SUBAPPLICATION Counter (* Subapplication Type *)
  (* Standard: 61499-2 *)
  (* Version 1.0, 2023-02-17, Franz *)
  IMPORT FBs::Counter::const::DefaultPool::AuxFunction2_MinusMinus;
  IMPORT FBs::Counter::const::DefaultPool::AuxFunction2_PlusPlus;
  IMPORT FBs::Counter::const::DefaultPool::Button_MinusMinus;
  IMPORT FBs::Counter::const::DefaultPool::Button_NextVT;
  IMPORT FBs::Counter::const::DefaultPool::Button_PlusPlus;
  IMPORT FBs::Counter::const::DefaultPool::Button_Reset_Gesamtzaehler;
  IMPORT FBs::Counter::const::DefaultPool::Button_Reset_Tageszaehler;
  IMPORT FBs::Counter::const::DefaultPool::NumberVariable_Gesamtzaehler;
  IMPORT FBs::Counter::const::DefaultPool::NumberVariable_Gesamtziel;
  IMPORT FBs::Counter::const::DefaultPool::NumberVariable_Tageszaehler;
  IMPORT FBs::Counter::const::DefaultPool::NumberVariable_Tagesziel;
  IMPORT FBs::Counter::const::DefaultPool::ObjectPointer_Gesamtziel;
  IMPORT FBs::Counter::const::DefaultPool::ObjectPointer_Tagesziel;
  IMPORT FBs::Counter::const::DefaultPool::SoftKey_MinusMinus;
  IMPORT FBs::Counter::const::DefaultPool::SoftKey_PlusPlus;
  IMPORT FBs::Counter::const::DefaultPool::SoftKey_Reset_Gesamtzaehler;
  IMPORT FBs::Counter::const::DefaultPool::SoftKey_Reset_Tageszaehler;
  IMPORT NVS_Keys::KEY_GESAMTZAEHLER;
  IMPORT NVS_Keys::KEY_GESAMTZIEL;
  IMPORT NVS_Keys::KEY_TAGESZAEHLER;
  IMPORT NVS_Keys::KEY_TAGESZIEL;
  IMPORT isobus::UT::io::Button::ButtonActivationCode::BT_RELEASED_UNLATCHED;
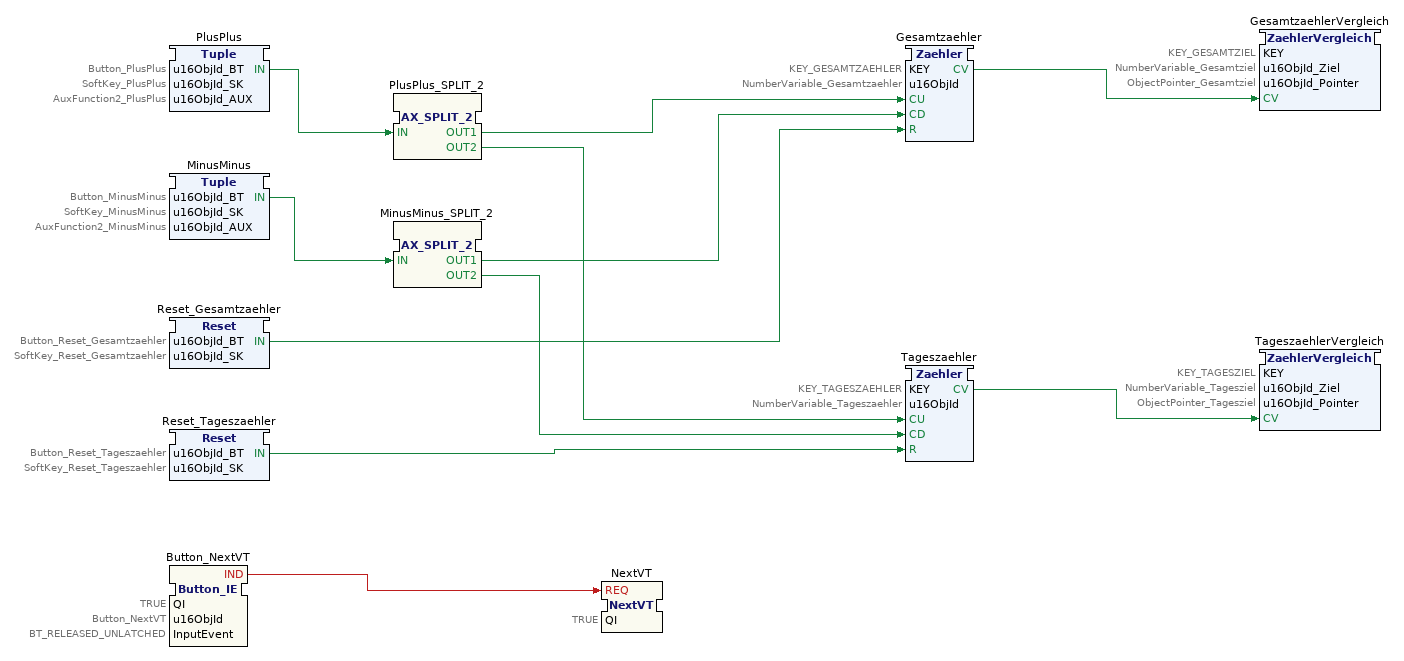
  FBS
    NextVT : isobus::UT::util::NextVT(QI := TRUE);
    Button_NextVT : isobus::UT::io::Button::Button_IE(QI := TRUE, u16ObjId := Button_NextVT, InputEvent := BT_RELEASED_UNLATCHED);
    PlusPlus_SPLIT_2 : adapter::events::unidirectional::AX_SPLIT_2;
    MinusMinus_SPLIT_2 : adapter::events::unidirectional::AX_SPLIT_2;
  END_FBS
  SUBAPPS
    MinusMinus : FBs::Counter::subs::Buttons::Tuple(u16ObjId_BT := Button_MinusMinus, u16ObjId_SK := SoftKey_MinusMinus, u16ObjId_AUX := AuxFunction2_MinusMinus);
    PlusPlus : FBs::Counter::subs::Buttons::Tuple(u16ObjId_BT := Button_PlusPlus, u16ObjId_SK := SoftKey_PlusPlus, u16ObjId_AUX := AuxFunction2_PlusPlus);
    Reset_Gesamtzaehler : FBs::Counter::subs::Buttons::Reset(u16ObjId_BT := Button_Reset_Gesamtzaehler, u16ObjId_SK := SoftKey_Reset_Gesamtzaehler);
    Reset_Tageszaehler : FBs::Counter::subs::Buttons::Reset(u16ObjId_BT := Button_Reset_Tageszaehler, u16ObjId_SK := SoftKey_Reset_Tageszaehler);
    Gesamtzaehler : FBs::Counter::subs::Zaehler::Zaehler(KEY := KEY_GESAMTZAEHLER, u16ObjId := NumberVariable_Gesamtzaehler);
    Tageszaehler : FBs::Counter::subs::Zaehler::Zaehler(KEY := KEY_TAGESZAEHLER, u16ObjId := NumberVariable_Tageszaehler);
    TageszaehlerVergleich : FBs::Counter::subs::Zaehler::ZaehlerVergleich(KEY := KEY_TAGESZIEL, u16ObjId_Ziel := NumberVariable_Tagesziel, u16ObjId_Pointer := ObjectPointer_Tagesziel);
    GesamtzaehlerVergleich : FBs::Counter::subs::Zaehler::ZaehlerVergleich(KEY := KEY_GESAMTZIEL, u16ObjId_Ziel := NumberVariable_Gesamtziel, u16ObjId_Pointer := ObjectPointer_Gesamtziel);
  END_SUBAPPS
  EVENT_CONNECTIONS
    Button_NextVT.IND TO NextVT.REQ;
  END_CONNECTIONS
  ADAPTER_CONNECTIONS
    PlusPlus.IN TO PlusPlus_SPLIT_2.IN;
    PlusPlus_SPLIT_2.OUT1 TO Gesamtzaehler.CU;
    PlusPlus_SPLIT_2.OUT2 TO Tageszaehler.CU;
    MinusMinus.IN TO MinusMinus_SPLIT_2.IN;
    MinusMinus_SPLIT_2.OUT1 TO Gesamtzaehler.CD;
    MinusMinus_SPLIT_2.OUT2 TO Tageszaehler.CD;
    Reset_Gesamtzaehler.IN TO Gesamtzaehler.R;
    Reset_Tageszaehler.IN TO Tageszaehler.R;
    Gesamtzaehler.CV TO GesamtzaehlerVergleich.CV;
    Tageszaehler.CV TO TageszaehlerVergleich.CV;
  END_CONNECTIONS
END_SUBAPPLICATION
